PROGRAM PRG_UpdateMotor
VAR
	resetMotor			: RS;
	
	gearingFactor		: INT := 460;
	gearingDivisor		: INT := 6;
	
	motorStartEvt		: DetectEvent;
	motorStopEvt		: DetectEvent;
	
END_VAR

resetMotor(	SET:= motorStartButton, RESET1 := motorStopButton, Q1 => motorStart);
motorTargetSpeed := (currentMotorSpeedSetting * gearingFactor)/gearingDivisor;

motorStartEvt(newSignalValue:= motorStartButton, detectLongClick := FALSE);
motorStopEvt(newSignalValue:= motorStopButton, detectLongClick := FALSE);

IF motorStartEvt.eventDetected = TASTEVT_PositiveEdge THEN
	motorStartButton := FALSE;
END_IF

IF motorStopEvt.eventDetected = TASTEVT_PositiveEdge THEN
	motorStopButton := FALSE;
END_IF

motorRpm := motorActualSpeed*gearingDivisor/gearingFactor;

IF motorStart THEN
	motorRunning := TRUE;
ELSE
	motorRunning := FALSE;
END_IF

(* TODO:
	--> what should happen when "RESET FAILURE" Button is pressed? 
*)

END_PROGRAM

(* stored: Version 1.1.0.1, ProductVersion 3.1.4022.7
   POU PRG_UpdateMotor: Id {07e9c43d-563b-405e-8f96-266c5264f4d5}, SpecialFunc None *)
